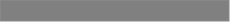
VISUALIZATION VISU_SUBSTRAT_NO_NUM  // 230x22
VAR_IN_OUT
	m_Input_MAP: STRUCT_MACHINE;
END_VAR
VAR_INPUT
	m_Input_NUM_CHAMBER : UDINT;
	m_Input_NUM_STATION : UDINT;
END_VAR
    Rectangle (0,0 228x20), invisible if: NOT m_Input_MAP.CHAMBER[m_Input_NUM_CHAMBER].STATION[m_Input_NUM_STATION].STATE_Unloaded
    Rectangle (0,0 228x20), invisible if: NOT m_Input_MAP.CHAMBER[m_Input_NUM_CHAMBER].STATION[m_Input_NUM_STATION].STATE_Loaded
    Rectangle (0,0 228x20), invisible if: m_Input_MAP.CHAMBER[m_Input_NUM_CHAMBER].STATION[m_Input_NUM_STATION].STATE_Loaded OR m_Input_MAP.CHAMBER[m_Input_NUM_CHAMBER].STATION[m_Input_NUM_STATION].STATE_Unloaded
END_VISUALIZATION

(* stored: Version 1.1.0.1, ProductVersion 3.1.4024.10
   Visu VISU_SUBSTRAT_NO_NUM: Id {56ead894-3a9b-4f3a-af7e-df68cedb2922} *)
